	{169.1274, 199.3721, 205.7021, 204.7051, 98.372, 208.1204, 137.3975},
	{170.4674, 199.3721, 240.7021, 205.7051, 98.372, 208.1204, 169.6812},
	{170.4674, 164.3721, 204.9021, 204.7051, 98.372, 173.1204, 169.6812},
	{168.7819, 165.8721, 206.4504, 204.7051, 99.372, 173.1204, 168.6812},
	{132.2819, 131.9512, 206.4504, 203.0196, 99.372, 173.1204, 168.6812},
	{131.2964, 133.4512, 206.4504, 203.0196, 98.032, 173.1204, 168.6812},
	{132.7964, 168.7504, 172.4812, 203.0196, 98.3875, 173.1204, 133.6812},
	{132.7964, 168.7504, 172.4812, 203.0196, 130.8084, 173.1204, 133.6812},
	{132.7964, 168.7504, 170.9812, 135.0812, 130.8084, 173.1204, 133.6812},
	{132.7964, 168.7504, 170.9812, 134.0812, 130.8084, 173.1204, 131.9957},
	{132.7964, 167.4204, 169.9504, 135.9912, 130.8084, 173.1204, 133.4957},
	{131.1109, 167.4204, 169.9504, 168.4121, 130.8084, 139.8512, 133.4957},
	{131.1109, 168.7504, 169.9504, 168.4121, 133.3484, 141.3512, 133.4957},
	{126.6509, 201.7196, 135.9812, 168.4121, 133.3484, 107.382, 133.4957},
	{162.9909, 201.7196, 169.9504, 168.4121, 133.3484, 107.382, 133.4957},
	{166.7509, 201.7196, 171.6359, 134.4429, 133.3484, 107.382, 133.4957},
	{169.9364, 201.7196, 171.6359, 134.4429, 133.3484, 107.382, 133.4957},
	{137.5155, 201.7196, 169.9504, 134.4429, 133.3484, 105.882, 133.4957},
	{137.5155, 201.7196, 171.6359, 134.4429, 133.3484, 105.182, 133.4957},
	{136.0155, 204.0596, 171.6359, 134.4429, 133.3484, 105.182, 133.4957},
	{136.0155, 204.0596, 171.6359, 134.4429, 133.3484, 105.182, 133.4957},
	{132.5455, 204.3904, 172.3359, 134.4429, 133.3484, 105.182, 133.4957},
	{136.0155, 203.0504, 206.3051, 134.4429, 132.7184, 105.882, 133.4957},
	{166.9364, 204.0359, 206.3051, 134.4429, 133.6884, 138.3512, 133.4957},
	{165.9364, 205.0359, 205.3051, 133.7429, 169.0339, 138.3512, 99.5265},
	{165.9364, 205.0359, 205.3051, 133.7429, 171.2339, 138.3512, 99.5265},
	{165.9364, 170.7359, 170.6359, 133.7429, 135.442, 172.9512, 99.5265},
	{165.9364, 170.7359, 170.6359, 133.7429, 137.1275, 171.4512, 97.841},
	{165.9364, 170.7359, 205.6359, 168.7429, 137.1275, 171.4512, 97.841},
	{165.9364, 170.7359, 205.6359, 168.7429, 137.1275, 171.4512, 133.471},
	{165.9364, 170.7359, 207.1359, 168.7429, 137.1275, 171.4512, 134.3255},
	{165.9364, 170.7359, 207.1359, 168.7429, 137.1275, 171.4512, 134.3255},
	{165.9364, 170.7359, 207.1359, 171.2812, 137.1275, 171.4512, 98.6955},
	{165.9364, 170.7359, 207.1359, 170.6357, 137.1275, 171.4512, 131.1164},
	{165.9364, 170.7359, 207.1359, 171.4665, 137.1275, 171.4512, 131.1164},
	{165.9364, 135.0812, 207.1359, 171.4665, 172.1275, 171.4512, 131.1164},
	{198.3573, 135.0812, 173.1667, 171.4665, 136.4975, 171.4512, 128.5764},
	{198.3573, 135.0812, 173.1667, 171.4665, 203.9184, 172.1512, 130.2619},
	{198.3573, 135.0812, 208.1667, 205.4265, 238.5484, 206.6349, 130.2619},
	{163.3573, 135.0812, 208.1667, 205.7812, 169.2484, 205.1349, 130.2619},
	{163.3573, 135.0812, 277.7659, 275.0496, 238.2176, 206.6349, 129.5619},
	{130.9364, 135.0812, 277.7659, 273.5496, 237.2176, 205.1349, 129.5219},
	{130.9364, 135.0812, 277.7659, 238.2504, 237.2176, 205.1349, 132.5474},
	{126.8364, 135.0812, 277.7659, 270.6713, 237.2176, 203.8049, 131.2174},
	{127.5364, 135.0812, 277.4204, 270.6713, 237.2176, 236.2258, 163.6383},
	{133.8364, 135.0812, 277.4204, 270.3313, 237.2176, 236.2258, 131.2174},
	{163.0056, 170.3804, 276.0804, 270.5168, 237.2176, 236.2258, 163.6383},
	{166.7656, 170.3804, 244.1022, 270.5168, 237.2176, 202.5566, 163.6383},
	{168.4511, 170.3804, 278.0714, 270.5168, 202.2176, 202.5566, 163.6383},
	{168.4511, 205.3804, 277.4259, 270.5168, 202.2176, 202.5566, 163.6383},
	{168.4511, 205.3804, 278.9259, 270.5168, 203.2576, 202.5566, 131.2174},
	{168.4511, 171.4112, 278.9259, 270.5168, 203.2576, 167.5566, 131.2174},
	{168.4511, 169.7257, 242.4259, 235.5168, 202.2176, 167.5566, 133.7574},
	{203.7503, 169.7257, 242.4259, 234.4768, 203.9031, 167.5566, 133.7574},
	{203.7503, 169.7257, 242.4259, 236.1623, 203.9031, 167.5566, 133.7574},
	{171.3294, 169.7257, 242.4259, 236.1623, 203.9031, 167.5566, 133.4174},
	{171.3294, 169.7257, 242.4259, 236.1623, 171.4822, 165.1711, 135.1029},
	{171.3294, 169.7257, 242.4259, 236.1623, 171.4822, 165.1711, 135.1029},
	{171.1694, 169.7257, 242.4259, 236.1623, 171.4822, 166.1711, 136.7884},
	{171.1694, 169.7257, 240.7404, 234.4768, 171.4822, 168.7111, 136.7884},
	{171.1694, 169.7257, 240.7404, 167.0559, 203.9031, 168.7111, 136.7884},
	{171.1694, 169.7257, 240.7404, 133.0867, 203.9031, 169.2594, 136.7884},
	{203.5903, 172.2657, 240.7404, 100.4575, 203.9031, 169.2594, 138.1339},
	{203.5903, 172.2657, 240.7404, 101.7975, 168.9031, 135.2902, 138.1339},
	{236.0112, 206.9349, 206.7712, 100.4575, 168.9031, 135.2902, 138.1884},
	{236.0112, 205.8949, 171.7712, 102.143, 134.9339, 135.2902, 139.6884},
	{236.0112, 137.112, 171.7712, 102.143, 134.9339, 135.2902, 174.3576}
};

// Singapore Prices
static REAL prices[49] [NUM_DAYS] = {

	{97.42, 74.13, 97.23, 135.8, 76.83, 76.83, 74.51},
	{91.02, 72.05, 86.03, 99.16, 75.35, 73.7, 67.84},
	{96.5, 69.26, 75.61, 77.19, 75.49, 68.11, 68.07},
	{85.71, 67.8, 73.04, 74.17, 73.12, 67.29, 68.37},
	{82.15, 66.81, 67.72, 72.15, 65.56, 66.07, 62.73},
	{76.81, 65.69, 67.26, 67.65, 64.77, 63.53, 62.09},
	{79.32, 64.69, 65.7, 66.95, 64.38, 63.51, 61.37},
	{70.9, 64.69, 64.92, 66.97, 64.28, 63.96, 60.38},
	{78.12, 64.37, 65.4, 67.02, 64.26, 63.5, 61.19},
	{80.53, 64.46, 65.65, 66.92, 64.36, 63.71, 60.13},
	{80.76, 65.5, 67, 67.75, 64.55, 64, 61.49},
	{83.05, 67.23, 72.43, 75.05, 64.81, 64.96, 61.37},
	{98.35, 69.89, 75.53, 77.89, 65.44, 64.93, 62.3},
	{110.12, 72.45, 85.04, 98.85, 66.77, 66.4, 62.47},
	{71.73, 64.45, 65.91, 68.47, 68.13, 67.86, 63.53},
	{79.58, 70.71, 71.29, 76.68, 67.91, 72.03, 63.02},
	{81.7, 73.99, 73.15, 105.23, 73.22, 70.72, 66.23},
	{82.15, 74.68, 78.59, 95.63, 76.78, 74.51, 67.33},
	{91.04, 82.67, 93.97, 105.34, 77.26, 77.02, 68.37},
	{97.54, 93.85, 124.65, 83.92, 85.82, 95.78, 70.4},
	{99.7, 125.15, 190.4, 94.34, 81.95, 129.48, 69.29},
	{146.29, 238.16, 250.55, 77.87, 95.21, 239.49, 70.35},
	{100.31, 224.94, 279.31, 76.84, 95.76, 254.78, 70.27},
	{98.44, 141.39, 201.3, 70.96, 94.65, 138.42, 70.39},
	{90.21, 100, 189.92, 68.93, 88.92, 114.4, 70.19},
	{91.72, 110.28, 249.42, 70.13, 88.84, 94.57, 71.01},
	{91.51, 159.82, 308.78, 72.38, 89.13, 92.31, 72.5},
	{91.67, 351.89, 347.53, 71.55, 86.44, 92.33, 72.89},
	{91.57, 352.79, 279.5, 69.62, 86.28, 86.84, 73.18},
	{86.31, 304.96, 240.44, 73.15, 86.37, 85.65, 72.48},
	{89.48, 241.81, 178.38, 77.08, 86.1, 84.6, 73.27},
	{86.32, 241.2, 140.48, 125.86, 78.77, 77.59, 73.29},
	{84.99, 241.27, 135.37, 99.95, 78.91, 76.91, 73.11},
	{84.86, 191.32, 98.9, 133.17, 78.03, 75.19, 72.46},
	{81.26, 102.62, 90.95, 97.58, 77.72, 75.02, 72.22},
	{83.17, 111.18, 76.08, 77.12, 91.99, 74.04, 75.12},
	{82.01, 87.08, 75.74, 76.41, 99.15, 74.61, 77.74},
	{83.12, 88.39, 94.26, 76.8, 92.51, 83.88, 77.98},
	{97.21, 98.43, 96.21, 81.65, 137.24, 96.98, 84.59},
	{99.82, 99.09, 104.69, 81.69, 178.22, 98.05, 97.38},
	{97.87, 101.06, 112.54, 77.33, 198.32, 105.6, 134.27},
	{191.42, 240.8, 239.95, 97.41, 222.7, 111.01, 141.57},
	{157.95, 240.73, 243.69, 77.14, 246.81, 96.42, 136.77},
	{124.96, 122.65, 179.28, 72.94, 138.33, 77.41, 124.99},
	{110.87, 97.61, 140.85, 73.1, 86.83, 79.65, 100.33},
	{78.32, 76.43, 99.22, 67.88, 81.91, 76.37, 83.32},
	{75.25, 74.22, 85.51, 68.13, 108.2, 74.55, 95.04},
	{71.28, 66.91, 76.99, 64.56, 77.62, 74.78, 79.81}

};

static REAL price[(48*7)+ 1]= {
	0,
	97.42,
	91.02,
	96.5,
	85.71,
	82.15,
	76.81,
	79.32,
	70.9,
	78.12,
	80.53,
	80.76,
	83.05,
	98.35,
	110.12,
	71.73,
	79.58,
	81.7,
	82.15,
	91.04,
	97.54,
	99.7,
	146.29,
	100.31,
	98.44,
	90.21,
	91.72,
	91.51,
	91.67,
	91.57,
	86.31,
	89.48,
	86.32,
	84.99,
	84.86,
	81.26,
	83.17,
	82.01,
	83.12,
	97.21,
	99.82,
	97.87,
	191.42,
	157.95,
	124.96,
	110.87,
	78.32,
	75.25,
	71.28,
	74.13,
	72.05,
	69.26,
	67.8,
	66.81,
	65.69,
	64.69,
	64.69,
	64.37,
	64.46,
	65.5,
	67.23,
	69.89,
	72.45,
	64.45,
	70.71,
	73.99,
	74.68,
	82.67,
	93.85,
	125.15,
	238.16,
	224.94,
	141.39,
	100,
	110.28,
	159.82,
	351.89,
	352.79,
	304.96,
	241.81,
	241.2,
	241.27,
	191.32,
	102.62,
	111.18,
	87.08,
	88.39,
	98.43,
	99.09,
	101.06,
	240.8,
	240.73,
	122.65,
	97.61,
	76.43,
	74.22,
	66.91,
	97.23,
	86.03,
	75.61,
	73.04,
	67.72,
	67.26,
	65.7,
	64.92,
	65.4,
	65.65,
	67,
	72.43,
	75.53,
	85.04,
	65.91,
	71.29,
	73.15,
	78.59,
	93.97,
	124.65,
	190.4,
	250.55,
	279.31,
	201.3,
	189.92,
	249.42,
	308.78,
	347.53,
	279.5,
	240.44,
	178.38,
	140.48,
	135.37,
	98.9,
	90.95,
	76.08,
	75.74,
	94.26,
	96.21,
	104.69,
	112.54,
	239.95,
	243.69,
	179.28,
	140.85,
	99.22,
	85.51,
	76.99,
	135.8,
	99.16,
	77.19,
	74.17,
	72.15,
	67.65,
	66.95,
	66.97,
	67.02,
	66.92,
	67.75,
	75.05,
	77.89,
	98.85,
	68.47,
	76.68,
	105.23,
	95.63,
	105.34,
	83.92,
	94.34,
	77.87,
	76.84,
	70.96,
	68.93,
	70.13,
	72.38,
	71.55,
	69.62,
	73.15,
	77.08,
	125.86,
	99.95,
	133.17,
	97.58,
	77.12,
	76.41,
	76.8,
	81.65,
	81.69,
	77.33,
	97.41,
	77.14,
	72.94,
	73.1,
	67.88,
	68.13,
	64.56,
	76.83,
	75.35,
	75.49,
	73.12,
	65.56,
	64.77,
	64.38,
	64.28,
	64.26,
	64.36,
	64.55,
	64.81,
	65.44,
	66.77,
	68.13,
	67.91,
	73.22,
	76.78,
	77.26,
	85.82,
	81.95,
	95.21,
	95.76,
	94.65,
	88.92,
	88.84,
	89.13,
	86.44,
	86.28,
	86.37,
	86.1,
	78.77,
	78.91,
	78.03,
	77.72,
	91.99,
	99.15,
	92.51,
	137.24,
	178.22,
	198.32,
	222.7,
	246.81,
	138.33,
	86.83,
	81.91,
	108.2,
	77.62,
	76.83,
	73.7,
	68.11,
	67.29,
	66.07,
	63.53,
	63.51,
	63.96,
	63.5,
	63.71,
	64,
	64.96,
	64.93,
	66.4,
	67.86,
	72.03,
	70.72,
	74.51,
	77.02,
	95.78,
	129.48,
	239.49,
	254.78,
	138.42,
	114.4,
	94.57,
	92.31,
	92.33,
	86.84,
	85.65,
	84.6,
	77.59,
	76.91,
	75.19,
	75.02,
	74.04,
	74.61,
	83.88,
	96.98,
	98.05,
	105.6,
	111.01,
	96.42,
	77.41,
	79.65,
	76.37,
	74.55,
	74.78,
	74.51,
	67.84,
	68.07,
	68.37,
	62.73,
	62.09,
	61.37,
	60.38,
	61.19,
	60.13,
	61.49,
	61.37,
	62.3,
	62.47,
	63.53,
	63.02,
	66.23,
	67.33,
	68.37,
	70.4,
	69.29,
	70.35,
	70.27,
	70.39,
	70.19,
	71.01,
	72.5,
	72.89,
	73.18,
	72.48,
	73.27,
	73.29,
	73.11,
	72.46,
	72.22,
	75.12,
	77.74,
	77.98,
	84.59,
	97.38,
	134.27,
	141.57,
	136.77,
	124.99,
	100.33,
	83.32,
	95.04,
	79.81
};

nb_samples = 8;
//int nb_samples_div_2 = nb_samples / 2;

	if (j < nb_samples/2){
	nb_samples = j;
	//nb_samples_div_2 = j / 2;
		}
	else if (j > 48*NUM_DAYS - 4){
	nb_samples = 48*NUM_DAYS - j+1;
	}
Std_forwrd_sum = 0;
Std_backwrd_sum = 0;
// SMA Calculation
    // foward sum
	for (int k = j + 1 ; k <= j+(nb_samples / 2);k++){
	Sma_forwrd += ( price[k]);
	}
	//Backward sum
	for (int k = j ; k > j-(nb_samples / 2); k--){
	Sma_backwrd += ( price[k]);
	}
	Sma_tot = (Sma_forwrd + Sma_backwrd)/ nb_samples ;// / nb_samples

//standard deviation Calculation
     // foward sum
	for (int k = j ; k <= j+nb_samples / 2;k++){

	Std_forwrd_sum += powf((price[k] - Sma_tot), 2);
	}
	//Backward sum
	for (int k = j + 1; k >= j-nb_samples / 2; k--){
	Std_backwrd_sum += powf((price[k] - Sma_tot), 2);
	}
	REAL sum1 = (Std_backwrd_sum + Std_forwrd_sum);
	if (nb_samples == 1){
	nb_samples = 2;
	}
	Std_dev = sqrt((sum1 )/ (nb_samples - 1 ));// / (nb_samples-1)

//put the code in here.
//DINT current_Minute = lol;

REAL current_price = prices[i][day];
REAL current_day = day;
REAL Demand = power_demand[lol][day];
//me->Minute = current_minute;

//printf("=====Current minute====, %d , %d \r\n",current_Minute, me->Minute );
//Setting Outputs of Input Block
//sifb_bfb_inputs_Algorithm1();
me->Minute = lol;
me->Price = current_price;
me->Demand_kWh =  power_demand[lol][day];
me->Day = current_day;

//	if (j==0){
//		me->Sma = 0;
//		me->Std_dev = 0;
//	}
//	else{


		me->Sma = Sma_tot;
		me->Std_dev = Std_dev;
//	}

printf("day = %f && Current minute is %d \r\n ", current_day, lol );
printf("Power = %f && Price is %f \r\n ", power_demand[lol][day], prices[i][day] );

if (lol%30 == 0 && lol != 0){
i++;
j++;
}

printf("Hello \r\n");
printf("%d", nb_samples);
printf("\r\n");
printf("%f", Sma_tot);
printf("\r\n");
printf("%f", Std_dev);
printf("\r\n");
printf("%d", j);
printf("\r\n");
//printf("%f",Std_forwrd_sum );
//printf("\r\n");

if (lol == 1440 && day == 6){ //End of Sunday

me->stop = 1;
//int hello = sayhello(2);
}

if (lol == 1440){
day++;
lol = 0;
i=0;
}
lol++;
  END_ALGORITHM
  ALGORITHM Algorithm1 IN C:

  END_ALGORITHM
END_FUNCTION_BLOCK
